FUNCTION_BLOCK TwoConCtlMulti (* Composite Function Block Type *)
  (* Standard: 61499-2 *)
  (* Version 0.2, 2003-12-05, JHC, Rockwell Automation, Renamed from NEWCOMPFB. *)
  (* Version 0.1, 2002-01-08, JHC, Rockwell Automation, Added DLY FB as example. *)
  (* Version 0.0, 2000-05-27, JHC, Rockwell Automation *)
  (* Compiler header: package fb.rt.cs725; *)
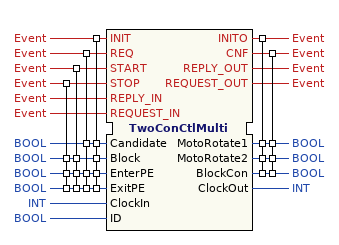
  EVENT_INPUT
    INIT WITH Candidate, Block, EnterPE, ExitPE; (* Initialization Request *)
    REQ WITH Candidate, EnterPE, ExitPE; (* Normal Execution Request *)
    START WITH Block, EnterPE, ExitPE;
    STOP WITH Block, EnterPE, ExitPE;
    REPLY_IN;
    REQUEST_IN;
  END_EVENT
  EVENT_OUTPUT
    INITO WITH MotoRotate1, MotoRotate2, BlockCon; (* Initialization Confirm *)
    CNF WITH MotoRotate1, MotoRotate2, BlockCon; (* Execution Confirmation *)
    REPLY_OUT;
    REQUEST_OUT;
  END_EVENT
  VAR_INPUT
    Candidate : BOOL;
    Block : BOOL;
    EnterPE : BOOL;
    ExitPE : BOOL;
    ClockIn : INT;
    ID : BOOL;
  END_VAR
  VAR_OUTPUT
    MotoRotate1 : BOOL;
    MotoRotate2 : BOOL;
    BlockCon : BOOL;
    ClockOut : INT;
  END_VAR
  FBS
    FC11 : ConveyorCTL(PE := 0, Block := 0, Candidate := 0);
    FC12 : ConveyorCTLMulti;
  END_FBS
  EVENT_CONNECTIONS
    INIT TO FC11.INIT;
    REQ TO FC11.REQ;
    FC12.INITO TO INITO;
    FC12.CNF TO CNF;
    REQ TO FC12.REQ;
    STOP TO FC12.CAS_STOP;
    START TO FC12.CAS_START;
    FC12.STOP TO FC11.CAS_STOP;
    FC12.START TO FC11.CAS_START;
    FC11.INITO TO FC12.INIT;
    REPLY_IN TO FC12.REPLY_IN;
    REQUEST_IN TO FC12.REQUEST_IN;
    FC12.REPLY_OUT TO REPLY_OUT;
    FC12.REQUEST_OUT TO REQUEST_OUT;
  END_CONNECTIONS
  DATA_CONNECTIONS
    Block TO FC12.Block;
    Candidate TO FC12.Candidate;
    FC12.BlockCon TO BlockCon;
    FC11.MotoRotate TO MotoRotate1;
    FC12.MotoRotate TO MotoRotate2;
    ExitPE TO FC12.ExitPE;
    EnterPE TO FC12.EnterPE;
    ID TO FC12.ID;
    ClockIn TO FC12.ClockIn;
    FC12.ClockOut TO ClockOut;
  END_CONNECTIONS
END_FUNCTION_BLOCK
